Staubli VAL3: PALLET.pjx

--- PALLET.pjx ---
Parameters version=s7.6.1 stackSize=5000 millimeterUnit=true
Program file=copy_it.pgx
Program file=link_all.pgx
Program file=link_it.pgx
Data file=PALLET.dtx
Library alias=saveData path=Disk://saveData/SAVEDATA.pjx
Type name=TrajPallet path=Disk://kernel/template/TrajPallet/TrajPallet.pjx
Type name=FrameItem path=Disk://kernel/template/FrameItem/FrameItem.pjx

--- PALLET.dtx ---
public TrajPallet tTraj{}

--- link_it.pgx ---
public program link_it(string x_sName)
begin
  // link ALL
  call link_all(x_sName)
  // put the base config
  tTraj[x_sName].tData[0].tSuper.toStop=true
  tTraj[x_sName].tData[0].tSuper.moveType=1
  tTraj[x_sName].tData[0].tSuper.comment=""
  tTraj[x_sName].trAppro[0]={0,0,-50,0,0,0}
  tTraj[x_sName].trAppro[1]={0,0,-50,0,0,0}
  tTraj[x_sName].trDepart[0]={0,0,-50,0,0,0}
  tTraj[x_sName].trDepart[1]={0,0,-50,0,0,0}
end
